(* CoDeSys 2.3.9.50 project: 6B.pr6 *)
(* Libraries: STANDARD.LB6 5.6.98 12:03:02 *)

(* POU MAIN, LD *)
PROGRAM MAIN
VAR
	T1: TOF;
	C1: CTU;
	reset AT %IX0.7: BOOL;
	reducedMOTOR AT %QX0.0: BOOL;
	normalMOTOR AT %QX0.1: BOOL;
	IncreasedMOTOR AT %QX0.2: BOOL;
	ACTUALResistance AT %IX0.1: BOOL;
	EXTRAResistance AT %IX0.2: BOOL;
	Processon AT %QX0.4: BOOL;
	Start AT %IX0.0: BOOL;
END_VAR
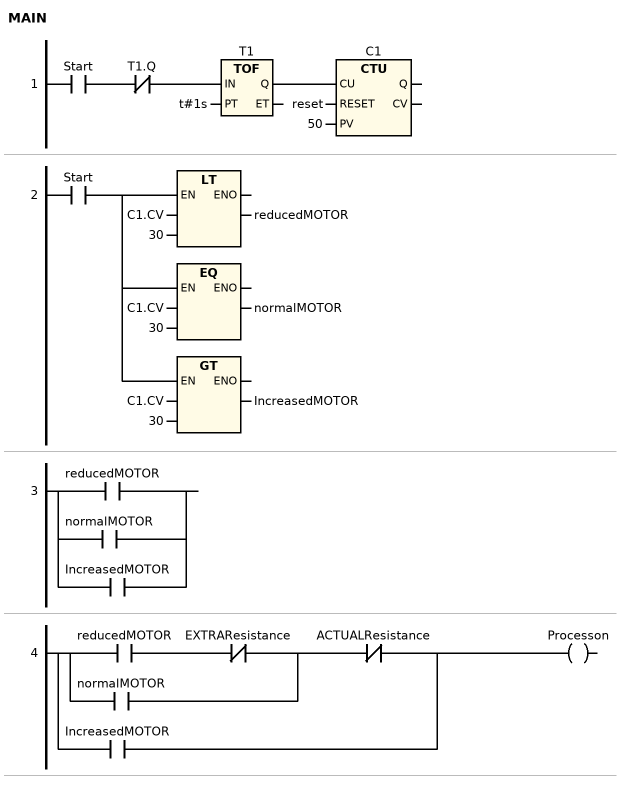
_LD_ (* Ladder Diagram *)
NETWORK 1
	[Start] - [/T1.Q] - T1:TOF(IN: *, PT: t#1s) - C1:CTU(CU: *, RESET: reset, PV: 50)
NETWORK 2
	[Start]
		EN --- LT(C1.CV, 30) => reducedMOTOR
		EN --- EQ(C1.CV, 30) => normalMOTOR
		EN --- GT(C1.CV, 30) => IncreasedMOTOR
NETWORK 3
	{ [reducedMOTOR] | [normalMOTOR] | [IncreasedMOTOR] }
NETWORK 4
	{ { [reducedMOTOR] - [/EXTRAResistance] | [normalMOTOR] } - [/ACTUALResistance] | [IncreasedMOTOR] } --- (Processon)
_END_LD_
(* the same logic as Structured Text *)
(* Network 1 *)
T1(IN := Start AND NOT T1.Q, PT := t#1s);
C1(CU := T1.Q, RESET := reset, PV := 50);
(* Network 2 *)
IF Start THEN
	reducedMOTOR := C1.CV < 30;
	normalMOTOR := C1.CV = 30;
	IncreasedMOTOR := C1.CV > 30;
END_IF;
(* Network 3 *)
(* Network 4 *)
Processon := (reducedMOTOR AND NOT EXTRAResistance OR normalMOTOR) AND NOT ACTUALResistance OR IncreasedMOTOR;
END_PROGRAM
